# B&R Automation Studio project ControllerSim
Automation Studio 4.9.2.46

## Configuration Simulation

CPU 5APC2200.AL14-000, AutomationRuntime D4.90, Build 4.1.2, Vc V4.72.2

### Hardware
```
5APC2200_AL14_000 : 5APC2200.AL14-000 v2.0.7.0
  Connector IF3:
    AssignedOperatingSystem = ARemb
    ActivateDevice = 1
  Connector IF4:
    AssignedOperatingSystem = ARemb
    ActivateDevice = 1
  Connector IF5:
    AssignedOperatingSystem = ARemb
  Connector IF6:
    AssignedOperatingSystem = ARemb
  ConfigurationID = ControllerSim_Simulation
  Simulation = 1
  ActivateOpcUa = 1
  OpcUa_AuthenticationSecurityPolicy_EnableNone = 1
  OpcUa_AuthenticationSecurityPolicy_EnableBasic128Rsa15 = 1
  OpcUaInformationModels_PV_Version = 2
```

## Logical view

### Global.typ - Global data types
```iecst
TYPE
	Enum1 :
		(
		Option1,
		Option2
		);
	Struct2 : 	STRUCT
		myFloat : REAL;
		myByte : USINT;
	END_STRUCT;
	Struct1 : 	STRUCT
		enum1 : Enum1;
		inner_struct : Struct2;
		myFloat : REAL;
		str : STRING[80];
		int_array : ARRAY[0..9]OF USINT;
	END_STRUCT;
END_TYPE
```

### Global.var - Global variables
```iecst
VAR
	e1 : Enum1;
	gCounter : USINT;
	flag : BOOL := TRUE;
	struct2 : Struct2;
	struct1 : Struct1;
END_VAR
```

### Program Logical/Program (IEC)

#### Main.st
```iecst
PROGRAM _INIT

	gCounter:=0;
	flag := TRUE;

	// just fill in some random data to read it at the PC side later
	struct1.enum1 := Option2;
	struct1.myFloat := 0.123;
	struct1.str := WSTRING_TO_STRING("FOO-BAR");
	FOR gCounter := 1 TO 9 DO
		struct1.int_array[gCounter] := struct1.int_array[gCounter] + gCounter;
	END_FOR;
	struct1.inner_struct.myByte := 100;
	struct1.inner_struct.myFloat := 3.1415;

	gCounter := 0;

	e1 := Option2;

	struct2.myByte := 42;
	struct2.myFloat := 2.345;
END_PROGRAM

PROGRAM _CYCLIC
	IF flag = TRUE THEN
		gCounter := gCounter + 1;
	END_IF
END_PROGRAM

PROGRAM _EXIT
	(* Insert code here *)

END_PROGRAM
```

Listed in the project but not available here: Logical/Libraries
